// TIA Portal V17 export
// export: Created 2024-08-07T21:44:14.5368505Z, ExportSetting WithDefaults, DisplayName Totally Integrated Automation Portal, DisplayVersion V17 Update 7, DisplayName TIA Portal Openness, DisplayVersion V17 Update 7, DisplayName TIA Portal Version Control Interface, DisplayVersion V17, DisplayName SINAMICS Startdrive Advanced, DisplayVersion V17 SP2, DisplayName SINAMICS Startdrive G110M, G120, G120C, G120D, G120P, G115D, DisplayVersion V17 SP2, DisplayName SINAMICS Startdrive G130, G150, S120, S150, SINAMICS MV, S210, DisplayVersion V17 SP2, DisplayName STEP 7 Professional, DisplayVersion V17 Update 7, DisplayName STEP 7 Safety, DisplayVersion V17 Update 6, DisplayName WinCC Advanced / Unified PC, DisplayVersion V17 Update 7
TYPE "UDT_Digiforce_receive"
// stored: IsFailsafeCompliant false
   STRUCT
      dataD : Struct
         Ready : Bool;
         OK : Bool;
         NOK : Bool;
         NOK_ONL : Bool;
         S1 : Bool;
         S2 : Bool;
         OK_STEST : Bool;
         MEAS_ACT : Bool;
         Strobe : Bool;
         Prog0 : Bool;
         Prog1 : Bool;
         Prog2 : Bool;
         reserve1 : Bool;
         reserve2 : Bool;
         reserve3 : Bool;
         reserve4 : Bool;
         Global_NOK : Bool;
         "Overload _NOK" : Bool;
         Window_1_NOK : Bool;
         Window_2_NOK : Bool;
         Window_3_NOK : Bool;
         Threshold_1_NOK : Bool;
         Threshold_2_NOK : Bool;
         Trapezoid_1_NOK : Bool;
         Trapezoid2_NOK : Bool;
         Envelope_NOK : Bool;
         "Measurement_w/o_READY" : Bool;
         USB_logging_error : Bool;
         reserve5 : Bool;
         reserve6 : Bool;
         reserve7 : Bool;
         reserve8 : Bool;
      END_STRUCT;
      dataA : Array[1..22] of Real;
   END_STRUCT;
END_TYPE
